{attribute 'GeneratedUsingTerminal: EL3621-0020-0016'}
{attribute addProperty BoxType "EL3621-0020-0016"}
{attribute addProperty Id "AI_InputsAT %I*AI_Inputs_4521310411WcStateAT %I*WcState_9091E0EB2InfoDataAT %I*InfoData_32EB74EA10"}
{attribute addProperty CRC "1887163282"}
{attribute addProperty Size "23"}
TYPE EL3621_707BD392 EXTENDS EtcSlaveTerminalBase_947E5A46 :
STRUCT
	{attribute addProperty Name "AI_Inputs"}
	AI_Inputs : AI_Inputs_45213104;
	{attribute addProperty Name "WcState"}
	WcState : WcState_9091E0EB;
	{attribute addProperty Name "InfoData"}
	InfoData : InfoData_32EB74EA;
END_STRUCT
END_TYPE

(* stored: Version 1.2.0.0, ProductVersion 3.1.4024.9
   DUT EL3621_707BD392: Id {5b7b0d87-93d7-4f22-a782-c41308f9c743} *)
